(* CODESYS project IC FLASHING FIX.project
   Title: Kitting Project
   Version: 0.0.0.0
   Author: lenovo

Project tree, tasks and I/O mapping:
  MyController : TM241CE40T/U, Schneider Electric, order no. TM241CE40T/U, version 4.0.6.18
    application Application
      libraries: Toolbox, 2.2.0.0 (Schneider Electric); SM3_Basic, 3.5.3.83 (3S - Smart Software Solutions GmbH); M241 PTOPWM, 1.0.0.23 (Schneider Electric)
      task MAST (cyclic, interval 20 ms, priority 15, watchdog 100 ms x 1) calls Tews, MyPOU, getIo, setIo, motor
      global variables GVL
      program motor [LD]
      program MyPOU [CFC]
      trace Trace (task MAST): iwModbusTCP_Slave_Device_Inputs_0
      program getIo [FBD]
      program Tews [LD]
      program setIo [FBD]
      program motor2 [FBD]
    DQ : Digital Outputs, Schneider Electric, version 4.0.6.18
        unmapped channels: QW0, QB1
    Ethernet_2 : Ethernet Network, Schneider Electric, version 4.0.6.18
        settings: IPAddress = [192, 168, 0, 11]; SubnetMask = [255, 255, 255, 0]; DeviceName = 'my_Device2'; WebServer = TRUE; FTP Server = TRUE; SoMachine Protocol = TRUE; Modbus Server = TRUE; NetManage Protocol = TRUE; SNMP protocol = TRUE
    Serial_Line_1 : Serial line, Schneider Electric, version 4.0.6.18
      SoMachine_Network_Manager : SoMachine-Network Manager, Schneider Electric, version 4.0.0.2
    Serial_Line_2 : Serial line, Schneider Electric, version 4.0.6.18
      Modbus_Manager : Modbus Manager, Schneider Electric, version 4.0.0.2
    DI : Digital Inputs, Schneider Electric, version 4.0.6.18
        unmapped channels: IDW0, IB1
    COM_Bus : COM bus, Schneider Electric, version 4.0.6.18
      Ethernet_1 : TM4ES4, Schneider Electric, order no. TM4ES4, version 1.0.0.10
          settings: IPAddress = [192, 168, 0, 10]; SubnetMask = [255, 255, 255, 0]; WebServer = TRUE; FTP Server = TRUE; SoMachine Protocol = TRUE; Modbus Server = TRUE; NetManage Protocol = TRUE; SNMP protocol = TRUE; Enable Routing = TRUE; WebVisu protocol = TRUE
    Pulse_Generators : Pulse Generators, Schneider Electric, version 4.0.6.18
    Counters : Counters, Schneider Electric, version 4.0.6.18
    Cartridge_1 : Cartridge, Schneider Electric, version 4.0.6.18
    Cartridge_2 : Cartridge, Schneider Electric, version 4.0.6.18
    IO_Bus : IO bus - TM3, Schneider Electric, version 4.0.6.18
      Module_1 : TM3DI16/G, Schneider Electric, order no. TM3DI16/G, version 1.0.1.4
          input  iwModule_1_IW0 : WORD  // IW0
          input  LDR_Sensor_OK_R_1 : BOOL  // IW0.I0
          input  LDR_Sensor_OK_R_2 : BOOL  // IW0.I1
          input  LDR_Sensor_OK_R_3 : BOOL  // IW0.I2
          input  LDR_Sensor_OK_R_4 : BOOL  // IW0.I3
          input  LDR_Sensor_OK_R_5 : BOOL  // IW0.I4
          input  LDR_Sensor_OK_R_6 : BOOL  // IW0.I5
          input  LDR_Sensor_OK_R_7 : BOOL  // IW0.I6
          input  LDR_Sensor_OK_R_8 : BOOL  // IW0.I7
          input  LDR_Sensor_NG_R_9 : BOOL  // IW0.I8
          input  LDR_Sensor_NG_R_10 : BOOL  // IW0.I9
          input  LDR_Sensor_NG_R_11 : BOOL  // IW0.I10
          input  LDR_Sensor_NG_R_12 : BOOL  // IW0.I11
          input  LDR_Sensor_NG_R_13 : BOOL  // IW0.I12
          input  LDR_Sensor_NG_R_14 : BOOL  // IW0.I13
          input  LDR_Sensor_NG_R_15 : BOOL  // IW0.I14
          input  LDR_Sensor_NG_R_16 : BOOL  // IW0.I15
      Module_2 : TM3DI16/G, Schneider Electric, order no. TM3DI16/G, version 1.0.1.4
          input  iwModule_2_IW0 : WORD  // IW0
          input  LDR_Sensor_OK_L_17 : BOOL  // IW0.I0
          input  LDR_Sensor_OK_L_18 : BOOL  // IW0.I1
          input  LDR_Sensor_OK_L_19 : BOOL  // IW0.I2
          input  LDR_Sensor_OK_L_20 : BOOL  // IW0.I3
          input  LDR_Sensor_OK_L_21 : BOOL  // IW0.I4
          input  LDR_Sensor_OK_L_22 : BOOL  // IW0.I5
          input  LDR_Sensor_OK_L_23 : BOOL  // IW0.I6
          input  LDR_Sensor_OK_L_24 : BOOL  // IW0.I7
          input  LDR_Sensor_NG_L_25 : BOOL  // IW0.I8
          input  LDR_Sensor_NG_L_26 : BOOL  // IW0.I9
          input  LDR_Sensor_NG_L_27 : BOOL  // IW0.I10
          input  LDR_Sensor_NG_L_28 : BOOL  // IW0.I11
          input  LDR_Sensor_NG_L_29 : BOOL  // IW0.I12
          input  LDR_Sensor_NG_L_30 : BOOL  // IW0.I13
          input  LDR_Sensor_NG_L_31 : BOOL  // IW0.I14
          input  LDR_Sensor_NG_L_32 : BOOL  // IW0.I15
      Module_3 : TM3DI32K, Schneider Electric, order no. TM3DI32K, version 1.0.1.3
          input  idwModule_3_ID0 : DWORD  // ID0
          input  PB_Start : BOOL  // ID0.I0
          input  Selector_Auto_Man : BOOL  // ID0.I1
          input  PB_Reset : BOOL  // ID0.I2
          input  PB_Stop : BOOL  // ID0.I3
          input  Smart_Relay : BOOL  // ID0.I4
          input  Program_lock_Right : BOOL  // ID0.I7
          input  Tray_Lock_right : BOOL  // ID0.I8
          input  Tray_Lock_left : BOOL  // ID0.I10
          input  Program_Lock_left : BOOL  // ID0.I11
          input  IC_Holder_Up_Left : BOOL  // ID0.I13
          input  IC_Holder_Down_left : BOOL  // ID0.I14
          input  Grip_IC_Tray_close : BOOL  // ID0.I15
          input  Grip_IC_Tray_open : BOOL  // ID0.I16
          input  IC_Holder_Up_right : BOOL  // ID0.I19
          input  IC_Holder_Down_right : BOOL  // ID0.I20
      Module_4 : TM3DI32K, Schneider Electric, order no. TM3DI32K, version 1.0.1.3
          input  idwModule_4_ID0 : DWORD  // ID0
          input  Data_Out_Vacuum_1 : BOOL  // ID0.I0
          input  Data_Out_Vacuum_2 : BOOL  // ID0.I1
          input  Data_Out_Vacuum_3 : BOOL  // ID0.I2
          input  Data_Out_Vacuum_4 : BOOL  // ID0.I3
          input  Data_Out_Vacuum_5 : BOOL  // ID0.I4
          input  Data_Out_Vacuum_6 : BOOL  // ID0.I5
          input  Data_Out_Vacuum_7 : BOOL  // ID0.I6
          input  Data_Out_Vacuum_8 : BOOL  // ID0.I7
          input  Data_Out_Vacuum_9 : BOOL  // ID0.I8
          input  Data_Out_Vacuum_10 : BOOL  // ID0.I9
          input  Data_Out_Vacuum_11 : BOOL  // ID0.I10
          input  Data_Out_Vacuum_12 : BOOL  // ID0.I11
          input  Data_Out_Vacuum_13 : BOOL  // ID0.I12
          input  Data_Out_Vacuum_14 : BOOL  // ID0.I13
          input  Data_Out_Vacuum_15 : BOOL  // ID0.I14
          input  Data_Out_Vacuum_16 : BOOL  // ID0.I15
      Module_5 : TM3DQ32TK, Schneider Electric, order no. TM3DQ32TK, version 1.0.1.3
          output Tower_Light_Red : BOOL  // QD0.Q0
          output Tower_Light_Yellow : BOOL  // QD0.Q1
          output Tower_Light_Green : BOOL  // QD0.Q2
          output Tower_Light_Blue : BOOL  // QD0.Q3
          output Buzzer : BOOL  // QD0.Q4
          output Emergency_Valve : BOOL  // QD0.Q5
          output Ring_Light : BOOL  // QD0.Q6
          output DIR_MOTOR : BOOL  // QD0.Q10
          output PULSE_MIN : BOOL  // QD0.Q11
          unmapped channels: QD0
      Module_6 : TM3DQ32TK, Schneider Electric, order no. TM3DQ32TK, version 1.0.1.3
          output Vacuum_1 : BOOL  // QD0.Q0
          output Vacuum_2 : BOOL  // QD0.Q1
          output Vacuum_3 : BOOL  // QD0.Q2
          output Vacuum_4 : BOOL  // QD0.Q3
          output Vacuum_5 : BOOL  // QD0.Q4
          output Vacuum_6 : BOOL  // QD0.Q5
          output Vacuum_7 : BOOL  // QD0.Q6
          output Vacuum_8 : BOOL  // QD0.Q7
          output Vacuum_9 : BOOL  // QD0.Q8
          output Vacuum_10 : BOOL  // QD0.Q9
          output Vacuum_11 : BOOL  // QD0.Q10
          output Vacuum_12 : BOOL  // QD0.Q11
          output Vacuum_13 : BOOL  // QD0.Q12
          output Vacuum_14 : BOOL  // QD0.Q13
          output Vacuum_15 : BOOL  // QD0.Q14
          output Vacuum_16 : BOOL  // QD0.Q15
          output Grip : BOOL  // QD0.Q16
          output Tray_Lock_right_Valve : BOOL  // QD0.Q17
          output Program_Lock_Right_valve : BOOL  // QD0.Q18
          output Program_Lock_Left_valve : BOOL  // QD0.Q19
          output Tray_Lock_Left_valve : BOOL  // QD0.Q20
          output IC_Hold_Left_valve : BOOL  // QD0.Q23
          output IC_Hold_Right_valve : BOOL  // QD0.Q24
          unmapped channels: QD0
*)

// MyController/Application/GVL
VAR_GLOBAL
END_VAR
VAR_GLOBAL
	out1 AT %QX0.0: BOOL;
    

END_VAR

// MyController/Application/Tews
PROGRAM Tews
VAR
END_VAR

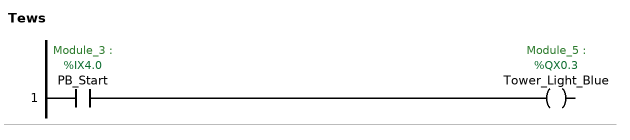
// NETWORK 1
//   PB_Start: Module_3 : | AT %IX4.0
//   Tower_Light_Blue: Module_5 : | AT %QX0.3
Tower_Light_Blue := PB_Start;

END_PROGRAM

// MyController/Application/MyPOU
PROGRAM MyPOU
VAR
END_VAR

END_PROGRAM

// MyController/Application/getIo
PROGRAM getIo
VAR

	READ_VAR_0: READ_VAR;
	ADDM_1: ADDM;
	addr_dss: ADDRESS;
	buffer_read: ARRAY[0..20] OF WORD;
	BLINK_0: BLINK;
	ADDR: POINTER TO BYTE;
	start:BOOL;
	WORD_AS_DWORD_0: WORD_AS_DWORD;
	WORD_AS_DWORD_1: WORD_AS_DWORD;
	inData AT %MW30:WORD;
	inData1 AT %MW31:WORD;
	inData2 AT %MW32:WORD;
	inData3 AT %MW33:WORD;
	inData4 AT %MW34:WORD;
	inData5 AT %MW35:WORD;
	inData6 AT %MW36:WORD;
	inData7 AT %MW37:WORD;
	inData8 AT %MW38:WORD;
	inData9 AT %MW39:WORD;
END_VAR

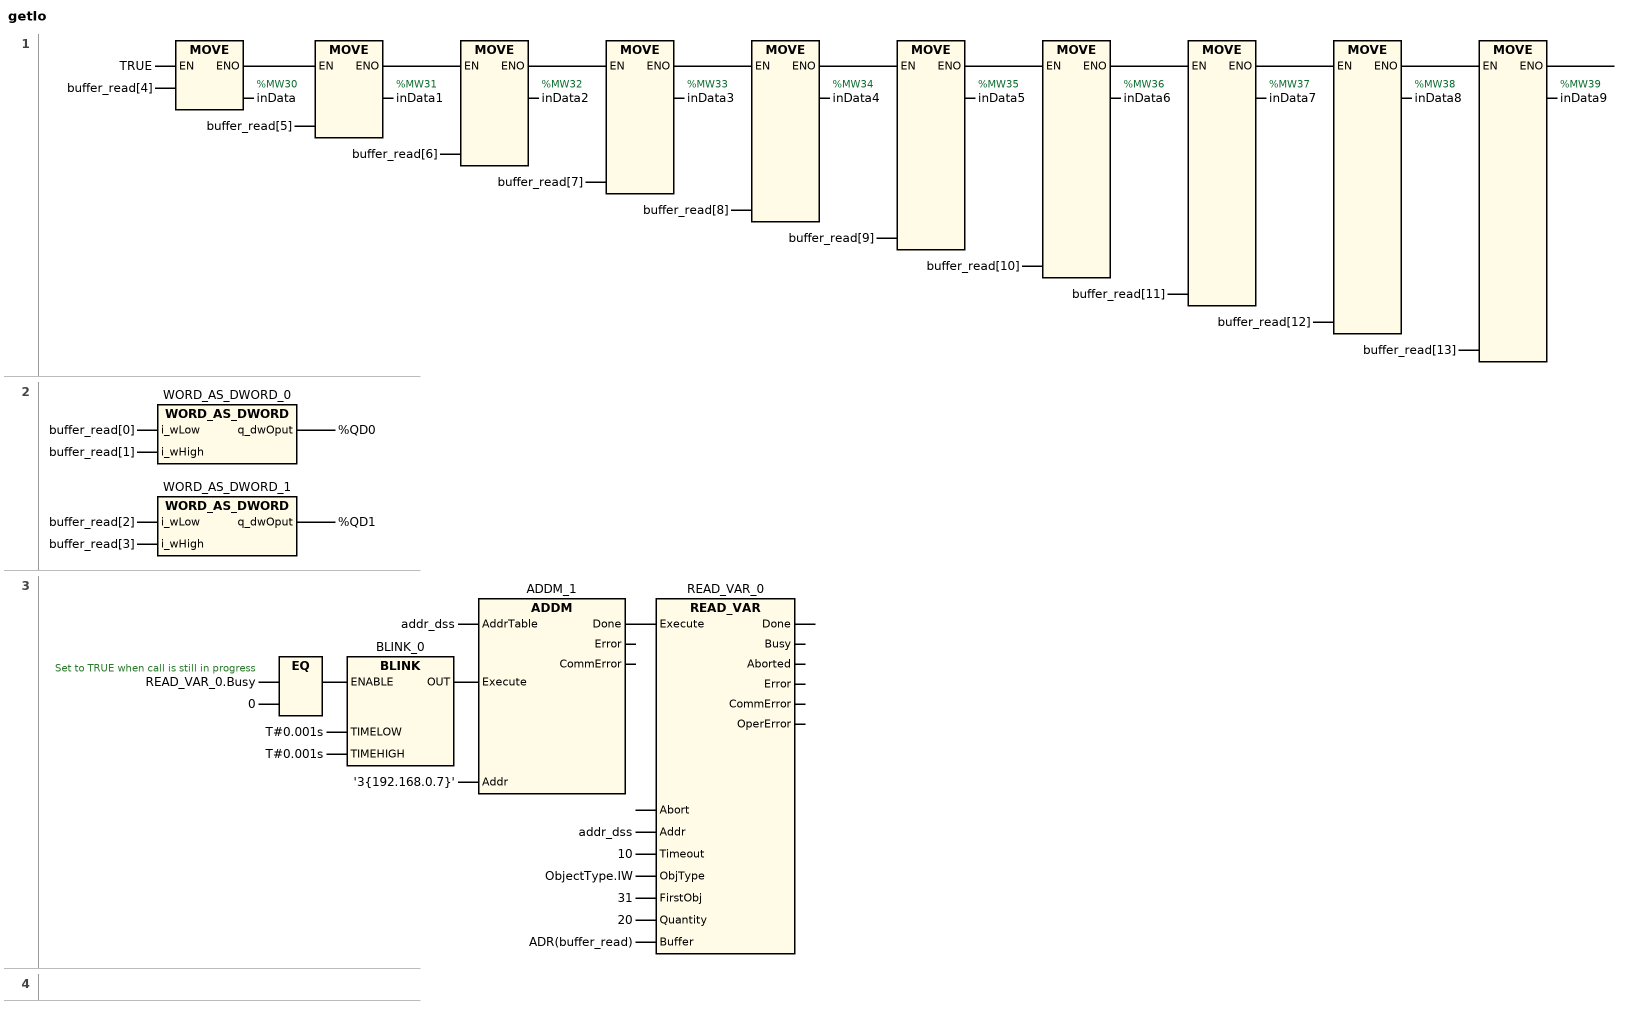
// NETWORK 1
//   inData: AT %MW30
//   inData1: AT %MW31
//   inData2: AT %MW32
//   inData3: AT %MW33
//   inData4: AT %MW34
//   inData5: AT %MW35
//   inData6: AT %MW36
//   inData7: AT %MW37
//   inData8: AT %MW38
//   inData9: AT %MW39
inData := buffer_read[4];
inData1 := buffer_read[5];
inData2 := buffer_read[6];
inData3 := buffer_read[7];
inData4 := buffer_read[8];
inData5 := buffer_read[9];
inData6 := buffer_read[10];
inData7 := buffer_read[11];
inData8 := buffer_read[12];
inData9 := buffer_read[13];

// NETWORK 2
WORD_AS_DWORD_0(i_wLow := buffer_read[0], i_wHigh := buffer_read[1]); // WORD_AS_DWORD
%QD0 := WORD_AS_DWORD_0.q_dwOput;
WORD_AS_DWORD_1(i_wLow := buffer_read[2], i_wHigh := buffer_read[3]); // WORD_AS_DWORD
%QD1 := WORD_AS_DWORD_1.q_dwOput;

// NETWORK 3
//   READ_VAR_0.Busy: Set to TRUE when call is still in progress
BLINK_0(ENABLE := READ_VAR_0.Busy = 0, TIMELOW := T#0.001s, TIMEHIGH := T#0.001s); // BLINK
ADDM_1(AddrTable := addr_dss, Execute := BLINK_0.OUT, Addr := '3{192.168.0.7}'); // ADDM
READ_VAR_0(
    Execute := ADDM_1.Done,
    Addr := addr_dss,
    Timeout := 10,
    ObjType := ObjectType.IW,
    FirstObj := 31,
    Quantity := 20,
    Buffer := ADR(buffer_read)); // READ_VAR

// NETWORK 4

END_PROGRAM

// MyController/Application/setIo
PROGRAM setIo
VAR
	WRITE_VAR_0: WRITE_VAR;
	ADDM_0: ADDM;
	BLINK_1: BLINK;
	addr_dss: ADDRESS;
	buffer_write: ARRAY[0..10] OF WORD;
	D1: DWORD_AS_WORD;
	outData AT %MW20:WORD;
	outData1 AT %MW21:WORD;
	outData2 AT %MW22:WORD;
	outData3 AT %MW23:WORD;
	outData4 AT %MW24:WORD;
	outData5 AT %MW25:WORD;
	outData6 AT %MW26:WORD;
	outData7 AT %MW27:WORD;
	outData8 AT %MW28:WORD;
	outData9 AT %MW29:WORD;

END_VAR

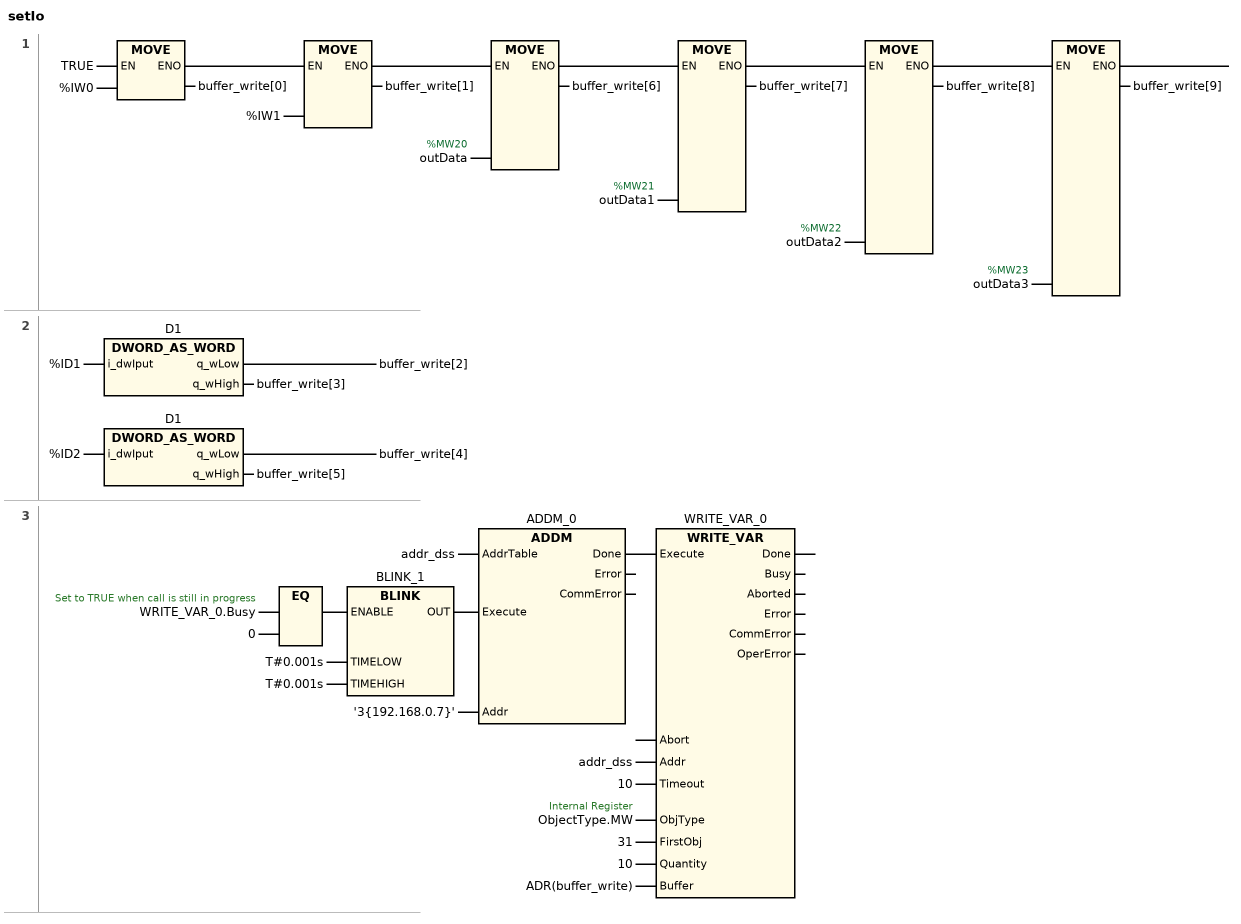
// NETWORK 1
//   outData: AT %MW20
//   outData1: AT %MW21
//   outData2: AT %MW22
//   outData3: AT %MW23
buffer_write[0] := %IW0;
buffer_write[1] := %IW1;
buffer_write[6] := outData;
buffer_write[7] := outData1;
buffer_write[8] := outData2;
buffer_write[9] := outData3;

// NETWORK 2
D1(i_dwIput := %ID1, q_wHigh => buffer_write[3]); // DWORD_AS_WORD
buffer_write[2] := D1.q_wLow;
D1(i_dwIput := %ID2, q_wHigh => buffer_write[5]); // DWORD_AS_WORD
buffer_write[4] := D1.q_wLow;

// NETWORK 3
//   WRITE_VAR_0.Busy: Set to TRUE when call is still in progress
//   ObjectType.MW: Internal Register
BLINK_1(ENABLE := WRITE_VAR_0.Busy = 0, TIMELOW := T#0.001s, TIMEHIGH := T#0.001s); // BLINK
ADDM_0(AddrTable := addr_dss, Execute := BLINK_1.OUT, Addr := '3{192.168.0.7}'); // ADDM
WRITE_VAR_0(
    Execute := ADDM_0.Done,
    Addr := addr_dss,
    Timeout := 10,
    ObjType := ObjectType.MW,
    FirstObj := 31,
    Quantity := 10,
    Buffer := ADR(buffer_write)); // WRITE_VAR

END_PROGRAM

// MyController/Application/motor
PROGRAM motor
VAR
	start: BOOL;
	t1: TON;
	
	reset: BOOL;
	t2: TON;
END_VAR

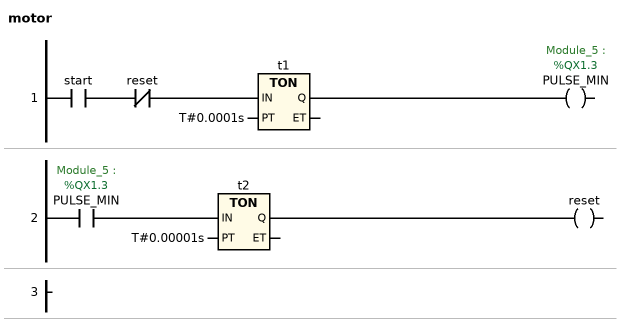
// NETWORK 1
//   PULSE_MIN: Module_5 : | AT %QX1.3
t1(IN := start AND NOT reset, PT := T#0.0001s); // TON
PULSE_MIN := t1.Q;

// NETWORK 2
//   PULSE_MIN: Module_5 : | AT %QX1.3
t2(IN := PULSE_MIN, PT := T#0.00001s); // TON
reset := t2.Q;

// NETWORK 3

END_PROGRAM

// MyController/Application/motor2
PROGRAM motor2
VAR
	mc_move: MC_MoveVelocity_PTO;
	
	PTO_X: AXIS_REF_PTO;
END_VAR

// NETWORK 1

END_PROGRAM
